Staubli VAL3: onF8Event.pgx

program onF8Event(bool& x_bSave[] (dimensions=1))
begin
  // look if the bButton is enable
  if bButton[7]
    //
    call insertIO(nSelected)
    x_bSave=true
  endIf
end
